// TIA Portal project "AX_Plc1516V3_CognexDataman" (V18)

(* hardware
DEVICE "S7-1500/ET200MP station_1"  S7-1500 station
   slot 0: "Rail_0"  Rack  6ES7 590-1***0-0AA0
   slot 1: "PLC_1"  CPU 1516-3 PN/DP  6ES7 516-3AP03-0AB0  V3.0
      slot 3: "CPU display_1"  6ES7591-1BA00-0AA0
      slot 32768: "PROFINET interface_1"  X1
         slot 32769: "Port_1"  X1 P1
         slot 32770: "Port_2"  X1 P2
      slot 33024: "PROFINET interface_2"  X2
         slot 33025: "Port_1"  X2 P1
      slot 33280: "DP interface_1"  X3
      slot 34817: "Virtual CP interface port_1"  Virtual CP interface port  Virtual CP interface port
DEVICE "GSD device_2"  GSD.Device.PN
   slot 0: "Rack"  Rack  V1.0
   slot 0: "10a1"  DataMan 280 CC-B  DMR-28x-xx  6.2.0
      slot 0: "DataMan 280 CC-B"  DataMan 280 CC-B
      slot 1: "Interface"  Interface
         slot 1: "Port 1"  Port 1
   slot 1: "Acquisition Control_1"  Acquisition Control
      slot 0: "Acquisition Control"  Acquisition Control
   slot 2: "Acquisition Status_1"  Acquisition Status
      slot 0: "Acquisition Status"  Acquisition Status
   slot 3: "Results Control_1"  Results Control
      slot 0: "Results Control"  Results Control
   slot 4: "Results Status_1"  Results Status
      slot 0: "Results Status"  Results Status
   slot 5: "Soft Event Control_1"  Soft Event Control
      slot 0: "Soft Event Control"  Soft Event Control
   slot 6: "User Data - 128 bytes_1"  User Data - 128 bytes
      slot 0: "User Data - 128 bytes"  User Data - 128 bytes
   slot 7: "Result Data - 128 bytes_1"  Result Data - 128 bytes
      slot 0: "Result Data - 128 bytes"  Result Data - 128 bytes
*)

// ===== PLC "PLC_1"  CPU 1516-3 PN/DP =====

ORGANIZATION_BLOCK "Main"   // OB1, LAD, ProgramCycle
TITLE = "Main Program Sweep (Cycle)"
{ S7_Optimized_Access := 'TRUE' }
VERSION : 0.1
   VAR_INPUT
      Initial_Call : Bool;   // Initial call of this OB
      Remanence : Bool;   // =True, if remanent data are available
   END_VAR
BEGIN
END_ORGANIZATION_BLOCK